// TIA Portal project "Inyectora_S7-1500" (V14)

(* hardware
DEVICE "S71500/ET200MP station_1"  S7-1500 station
   slot 0: "Perfil soporte_0"  Rack  6ES7 590-1***0-0AA0
   slot 1: "Inyectora"  CPU 1511-1 PN  6ES7 511-1AK01-0AB0  V2.1
      slot 3: "Display de la CPU_1"  6ES7591-1AA00-0AA0
   slot 2: "DI 16x24VDC BA_1"  DI 16x24VDC BA  6ES7 521-1BH10-0AA0  V1.0
   slot 3: "DQ 8x24VDC/2A HF_1"  DQ 8x24VDC/2A HF  6ES7 522-1BF00-0AB0  V2.1
   slot 4: "AI 8xU/I/RTD/TC ST_1"  AI 8xU/I/RTD/TC ST  6ES7 531-7KF00-0AB0  V2.1
   slot 5: "AI 8xU/I/RTD/TC ST_2"  AI 8xU/I/RTD/TC ST  6ES7 531-7KF00-0AB0  V2.1
   slot 6: "AI 8xU/I/RTD/TC ST_4"  AI 8xU/I/RTD/TC ST  6ES7 531-7KF00-0AB0  V2.1
   slot 7: "AI 8xU/I/RTD/TC ST_5"  AI 8xU/I/RTD/TC ST  6ES7 531-7KF00-0AB0  V2.1
   slot 8: "AQ 8xU/I HS_1"  AQ 8xU/I HS  6ES7 532-5HF00-0AB0  V2.1
   slot 9: "AQ 8xU/I HS_2"  AQ 8xU/I HS  6ES7 532-5HF00-0AB0  V2.1
*)

// ===== PLC "Inyectora"  CPU 1511-1 PN =====

VAR_GLOBAL   // PLC tag table "Tabla de variables estándar"
   "System_Byte" AT %MB1 : Byte;
   "FirstScan" AT %M1.0 : Bool;
   "DiagStatusUpdate" AT %M1.1 : Bool;
   "AlwaysTRUE" AT %M1.2 : Bool;
   "AlwaysFALSE" AT %M1.3 : Bool;
   "System_Byte(1)" AT %MB1 : Byte;
   "Clock_Byte" AT %MB0 : Byte;
   "Clock_10Hz" AT %M0.0 : Bool;
   "Clock_5Hz" AT %M0.1 : Bool;
   "Clock_2.5Hz" AT %M0.2 : Bool;
   "Clock_2Hz" AT %M0.3 : Bool;
   "Clock_1.25Hz" AT %M0.4 : Bool;
   "Clock_1Hz" AT %M0.5 : Bool;
   "Clock_0.625Hz" AT %M0.6 : Bool;
   "Clock_0.5Hz" AT %M0.7 : Bool;
   "DI_Selectora_Calentar" AT %I1.3 : Bool;   // Selectora 0=OFF; 1=ON
   "AQ_S_RETROCESO_CARRO" AT %QW104 : Int;
END_VAR

VAR_GLOBAL   // PLC tag table "DI"
   "DI_R_CARGA" AT %I0.2 : Bool;   // Recorridos de carga
   "DI_R_SUCCION" AT %I0.1 : Bool;   // Recorrido de succión
   "DI_S_PUERTA" AT %I0.0 : Bool;   // Seguridad de las puertas
   "DI_E_Local" AT %I0.3 : Bool;   // Parada de Emergencia desde el Tablero LOCAL
   "DI_E_Remoto" AT %I0.4 : Bool;   // Parada de Emergencia desde el Tablero Remoto
   "DI_Selectora_M" AT %I0.5 : Bool;   // Selectora MANUAL 0=OFF; 1=ON
   "DI_Selectora_S" AT %I0.6 : Bool;   // Selectora SEMIAUTOMATICO 0=OFF; 1=ON
   "DI_Selectora_A" AT %I0.7 : Bool;   // Selectora AUTOMATICO 0=OFF; 1=ON
   "DI_Arranque_L" AT %I1.0 : Bool;   // Boton de arranque del tablero LOCAL
   "DI_Parada_L" AT %I1.1 : Bool;   // Boton de parada del tablero LOCAL
   "DI_Selectora_LR" AT %I1.2 : Bool;   // Selectora 0=LOCAL; 1=REMOTO
END_VAR

VAR_GLOBAL   // PLC tag table "AI"
   "AI_P_HYD_INYECCION" AT %IW10 : Int;   // Presión Hidráulica de inyecc
   "AI_P_CE_MOLDE" AT %IW12 : Int;   // Presión de cierre de molde
   "AI_P_AP_MOLDE" AT %IW14 : Int;   // Presión de apertura de molde
   "AI_P_EXP_PIEZA" AT %IW16 : Int;   // Presión de expulsión de las piezas
   "AI_P_SUCCION" AT %IW18 : Int;   // Presión de succión
   "AI_P_MOV_CARRO" AT %IW20 : Int;   // Presión de movimiento carro
   "AI_P_GENERAL" AT %IW22 : Int;   // Presión general
   "AI_V_CARGA" AT %IW24 : Int;   // Velocidad de carga 0..100
   "AI_V_INYECCION" AT %IW30 : Int;   // Velocidad de inyección
   "AI_V_AP_MOLDE" AT %IW32 : Int;   // Velocidad de apertura de molde
   "AI_V_CE_MOLDE" AT %IW34 : Int;   // Velocidad de cierre de molde
   "AI_V_EXP_AVANCE" AT %IW36 : Int;   // Velocidad de expulsión avance
   "AI_V_EXP_RETROCESO" AT %IW38 : Int;   // Velocidad de expulsión retroceso
   "AI_V_CARRO" AT %IW40 : Int;   // Velocidad del carro
   "AI_V_SUCCION" AT %IW42 : Int;   // Velocidad de succión
   "AI_T_Z_ALIMENTACION" AT %IW44 : Int;   // Zona de Alimentación-real
   "T_Z_PLASTIFICACION" AT %IW90 : Int;   // Zona de Plastificación
   "T_Z_DOSIFICACION" AT %IW92 : Int;   // Zona de Dosifacion
   "T_Z_BOQUILLA" AT %IW94 : Int;   // Zona de Boquilla
   "T_MOLDE" AT %IW96 : Int;   // Temperatura del Molde
   "T_ACEITE_HYD" AT %IW98 : Int;   // Temperatura del Aceite Hidráulico
   "T_GABINETE" AT %IW100 : Int;   // Temperatura del Gabinete eléctrico
   "R_AV_INYECTOR" AT %IW102 : Int;   // Recorridos de avance inyector
   "R_AP_MOLDE" AT %IW104 : Int;   // Recorrido apertura del molde
   "AI_R_CE_MOLDE" AT %IW70 : Int;   // Recorrido cierre del molde
   "AI_R_CARRO" AT %IW72 : Int;   // Recorrido del carro
   "AI_R_EXPULSION" AT %IW74 : Int;   // Recorrido de la expulsión
END_VAR

VAR_GLOBAL   // PLC tag table "DQ"
   "DQ_VENTILADOR_GABINETE" AT %Q0.0 : Bool;
   "DQ_Z_ALIMENTACION" AT %Q0.1 : Bool;
   "DQ_Z_PLASTIFICACION" AT %Q0.2 : Bool;
   "DQ_Z_DOSIFICACION" AT %Q0.3 : Bool;
   "DQ_Z_BOQUILLA" AT %Q0.4 : Bool;
   "DQ_VENTILADOR" AT %Q0.5 : Bool;
END_VAR

VAR_GLOBAL   // PLC tag table "AQ"
   "AQ_S_INYECCION" AT %QW90 : Int;   // Solenoide de inyección
   "AQ_S_SUCCION" AT %QW92 : Int;   // Solenoide de succión
   "AQ_S_CARGA" AT %QW94 : Int;   // Solenoide de carga
   "AQ_S_EXPULSION" AT %QW96 : Int;   // Solenoide de Expulsión
   "AQ_S_AVANCE_CARRO" AT %QW98 : Int;   // Solenoide de movimiento de Carro
   "AQ_S_P_GENERAL" AT %QW100 : Int;   // Solenoide de presión General
   "AQ_S_R_CAUDAL" AT %QW102 : Int;   // Selenoide regulador de caudal
   "AQ_S_NOYO2" AT %QW110 : Int;   // Solenoide Noyo
   "AQ_S_NOYO3" AT %QW112 : Int;   // Solenoide Noyo
END_VAR

TYPE "Mediciones"
   STRUCT
      Medicion : Array[1..10] of Real;
   END_STRUCT;
END_TYPE

DATA_BLOCK "DB_Sistema"   // DB1
{ S7_Optimized_Access := 'TRUE' }
VERSION : 0.1
   VAR
      Lecturas : Struct   // Lecturas Procesadas
         Temperatura : Struct   // Lecturas de Temperatura, escaladas y normalizadas.
            Alimentacion : Real;   // Valor de Temperatura en la Zona de Alimentacion, ya normalizada y escalada.
            Plastificacion : Real;   // Valor de Temperatura en la Zona de Plastificacion, ya normalizada y escalada.
            Dosificacion : Real;   // Valor de Temperatura en la Zona de Dosificacion, ya normalizada y escalada.
            Boquilla : Real;   // Valor de Temperatura en la Zona de Boquilla, ya normalizada y escalada.
            Molde : Real;   // Valor de Temperatura del Molde, ya normalizada y escalada.
            Aceite : Real;   // Valor de Temperatura en el Aceite, ya normalizada y escalada.
            Gabinete : Real;   // Valor de Temperatura en el Gabinete, ya normalizada y escalada.
         END_STRUCT;
         Velocidad : Struct   // Lecturas de Velocidad, escalados y normalizados.
            Carga : Real;
            Inyeccion : Real;
            Apertura_Molde : Real;
            Cierre_Molde : Real;
            Expulsion_Avance : Real;
            Expulsion_Retroceso : Real;
            Carro : Real;
            Succion : Real;
         END_STRUCT;
         Recorrido : Struct   // Lecturas de Recorrido, escalados y normalizados.
            Avance_Inyector : Real;
            Apertura_Molde : Real;
            Cierre_Molde : Real;
            Carro : Real;
            Expulsion : Real;
         END_STRUCT;
         Presion : Struct   // Lecturas de Presiones, escaladas y normalizadas.
            Hidraulica_inyeccion : Real;
            Cierre_Molde : Real;
            Apertura_Molde : Real;
            Expulsion_Pieza : Real;
            Succion : Real;
            Movimiento_Carro : Real;
            General : Real;
            Seguridad_Molde : Real;
         END_STRUCT;
         Nivel_Tolva : Real;   // Lectura de Nivel, escalada y normalizada.
      END_STRUCT;
      Consigna : Struct   // Establecimiento de los Set Points
         Temperatura : Struct
            Alimentacion : Real;
            Plastificacion : Real;
            Dosificacion : Real;
            Boquilla : Real;
            Molde : Real;
            Aceite : Real;
            Gabinete : Real;
         END_STRUCT;
         Velocidad : Struct
            Carga : Real;
            Inyeccion : Real;
            Apertura_Molde : Real;
            Cierre_Molde : Real;
            Expulsion_Avance : Real;
            Expulsion_Retroceso : Real;
            Carro : Real;
            Succion : Real;
         END_STRUCT;
         Recorrido : Struct
            Avance_Inyector : Bool;
            Apertura_Molde : Bool;
            Cierre_Molde : Bool;
            Carro : Bool;
            Expulsion : Bool;
         END_STRUCT;
         Presion : Struct
            Hidraulica_inyeccion : Bool;
            Cierre_Molde : Bool;
            Apertura_Molde : Bool;
            Expulsion_Pieza : Bool;
            Succion : Bool;
            Movimiento_Carro : Bool;
            General : Bool;
            Seguridad_Molde : Bool;
         END_STRUCT;
         Tiempo : Struct
            Inyeccion : Real;
            Carga : Real;
            Curado : Real;
            Apertura_Molde : Real;
            Cierre_Molde : Real;
            Expulsion : Real;
            Retencion_Expulsion : Real;
            Reciclo : Real;
            Succion : Real;
            Carro : Real;
            Ciclo_Completo : Real;
         END_STRUCT;
      END_STRUCT;
      HMI : Struct   // Comandos del HMI
         CMD_Parada : Bool;   // Boton Parada HMI
         CMD_Arranque : Bool;   // Boton Arranque HMI
      END_STRUCT;
      Marcas : Struct   // Marcas para valores intermedios
         Selenoides : Struct
            Inyeccion : Bool;
            Succion : Bool;
            Carga : Bool;
            Expulsion : Bool;
            Avance_Carro : Bool;
            Retroceso_Carro : Bool;
            Presion_General : Bool;
            Regulador_Caudal : Bool;
            Noyo : Array[1..3] of Bool;
         END_STRUCT;
      END_STRUCT;
      Seguridad : Struct   // Marcas para control de seguridad
         Parada_Controlada : Bool;
         Parada_Emergencia : Bool;
      END_STRUCT;
      Paso : Array[1..10] of Bool;   // Marcas de pasos a seguir en la secuencia
   END_VAR
BEGIN
END_DATA_BLOCK

DATA_BLOCK "Valvula_Proporcional_1"   // DB5
{ S7_Optimized_Access := 'TRUE' }
VERSION : 0.1
// stored: InstanceOfName Valvula_Proporcional
"Valvula_Proporcional"
BEGIN
END_DATA_BLOCK

FUNCTION_BLOCK "Filtro"   // FB1, LAD
{ S7_Optimized_Access := 'TRUE' }
VERSION : 0.1
   VAR_INPUT
      Medicion : Real;
   END_VAR
   VAR_OUTPUT
      Valor_filtrado : Real;
   END_VAR
   VAR
      Mediciones : "Mediciones";
   END_VAR
   VAR_TEMP
      Sumatoria : Real;
   END_VAR
   VAR CONSTANT
      Divisior : Real := 10.0;
   END_VAR
BEGIN

REGION Network 1
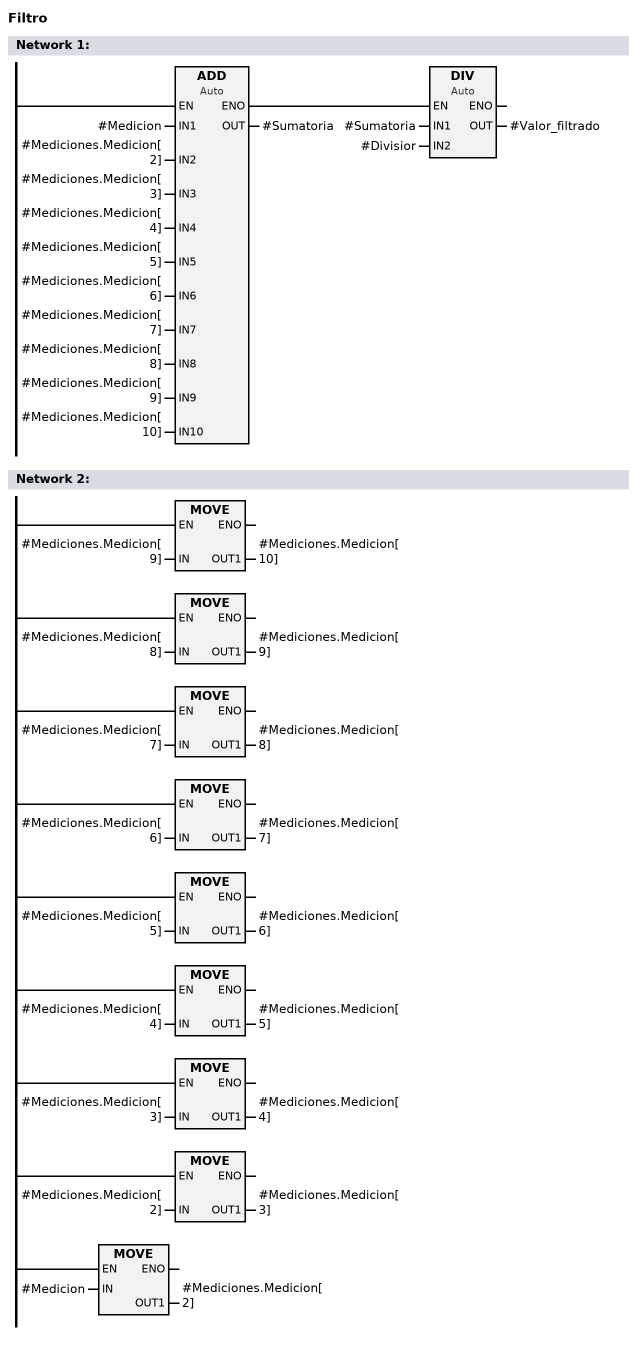
   RUNG wire#powerrail
      Add(in1 := #Medicion, in2 := #Mediciones.Medicion[2], in3 := #Mediciones.Medicion[3], in4 := #Mediciones.Medicion[4], in5 := #Mediciones.Medicion[5], in6 := #Mediciones.Medicion[6], in7 := #Mediciones.Medicion[7], in8 := #Mediciones.Medicion[8], in9 := #Mediciones.Medicion[9], in10 := #Mediciones.Medicion[10], out => #Sumatoria)
      Div(in1 := #Sumatoria, in2 := #Divisior, out => #Valor_filtrado)
   END_RUNG
   // the same network as SCL:
   #Sumatoria := #Medicion + #Mediciones.Medicion[2] + #Mediciones.Medicion[3] + #Mediciones.Medicion[4] + #Mediciones.Medicion[5] + #Mediciones.Medicion[6] + #Mediciones.Medicion[7] + #Mediciones.Medicion[8] + #Mediciones.Medicion[9] + #Mediciones.Medicion[10];
   #Valor_filtrado := #Sumatoria / #Divisior;
END_REGION

REGION Network 2
   RUNG wire#powerrail
      Move(in := #Mediciones.Medicion[9], out1 => #Mediciones.Medicion[10])
   END_RUNG
   RUNG wire#powerrail
      Move(in := #Mediciones.Medicion[8], out1 => #Mediciones.Medicion[9])
   END_RUNG
   RUNG wire#powerrail
      Move(in := #Mediciones.Medicion[7], out1 => #Mediciones.Medicion[8])
   END_RUNG
   RUNG wire#powerrail
      Move(in := #Mediciones.Medicion[6], out1 => #Mediciones.Medicion[7])
   END_RUNG
   RUNG wire#powerrail
      Move(in := #Mediciones.Medicion[5], out1 => #Mediciones.Medicion[6])
   END_RUNG
   RUNG wire#powerrail
      Move(in := #Mediciones.Medicion[4], out1 => #Mediciones.Medicion[5])
   END_RUNG
   RUNG wire#powerrail
      Move(in := #Mediciones.Medicion[3], out1 => #Mediciones.Medicion[4])
   END_RUNG
   RUNG wire#powerrail
      Move(in := #Mediciones.Medicion[2], out1 => #Mediciones.Medicion[3])
   END_RUNG
   RUNG wire#powerrail
      Move(in := #Medicion, out1 => #Mediciones.Medicion[2])
   END_RUNG
   // the same network as SCL:
   #Mediciones.Medicion[10] := #Mediciones.Medicion[9];
   #Mediciones.Medicion[9] := #Mediciones.Medicion[8];
   #Mediciones.Medicion[8] := #Mediciones.Medicion[7];
   #Mediciones.Medicion[7] := #Mediciones.Medicion[6];
   #Mediciones.Medicion[6] := #Mediciones.Medicion[5];
   #Mediciones.Medicion[5] := #Mediciones.Medicion[4];
   #Mediciones.Medicion[4] := #Mediciones.Medicion[3];
   #Mediciones.Medicion[3] := #Mediciones.Medicion[2];
   #Mediciones.Medicion[2] := #Medicion;
END_REGION
END_FUNCTION_BLOCK

FUNCTION_BLOCK "Valvula_Proporcional"   // FB2, LAD
{ S7_Optimized_Access := 'TRUE' }
VERSION : 0.1
   VAR_INPUT
      Consigna_Velocidad : Real;
      Posicion : Real;
   END_VAR
   VAR_OUTPUT
      Salida : Real;
   END_VAR
   VAR
      Captura_Posicion : Real;
   END_VAR
   VAR_TEMP
      PID_Salida : Real;
      Velocidad : Real;
      Porciento : Real;
   END_VAR
   VAR CONSTANT
      Divisor : Real := 0.01;   // La diferencia de tiempo es constante, se activa por una interrupcion ciclica
   END_VAR
BEGIN

REGION Network 1
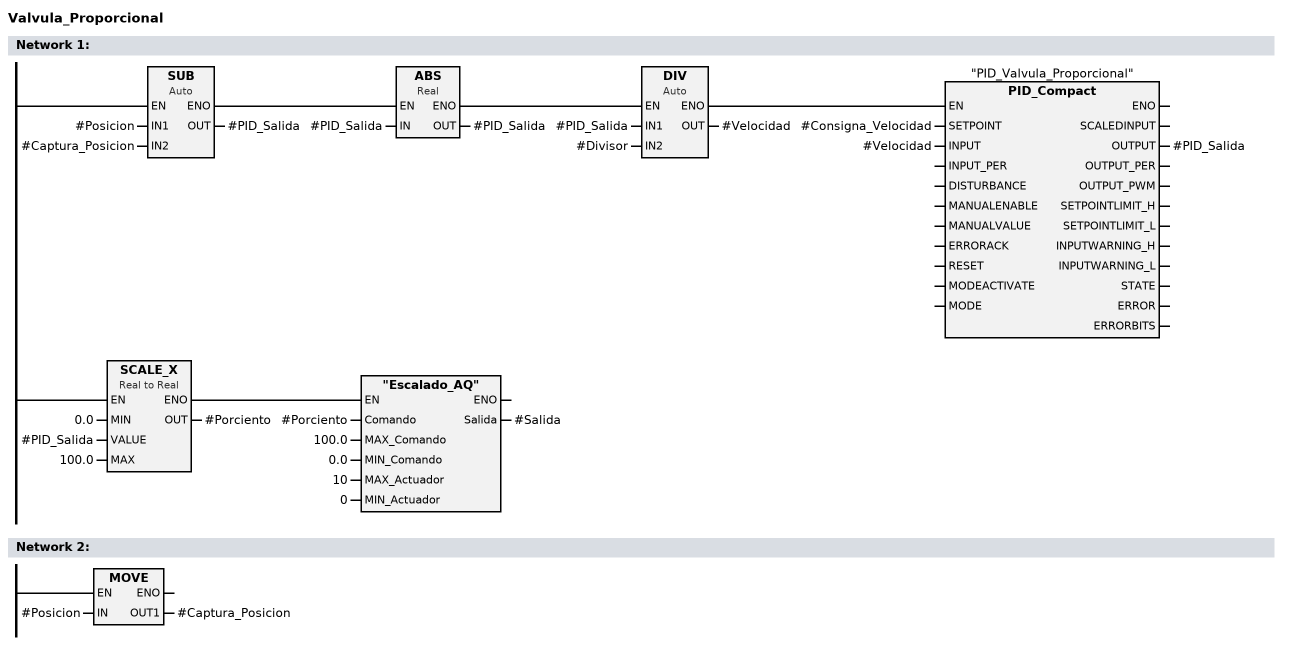
   #PID_Salida := #Posicion - #Captura_Posicion;
   #PID_Salida := ABS(#PID_Salida);
   #Velocidad := #PID_Salida / #Divisor;
   "PID_Valvula_Proporcional"(Setpoint := #Consigna_Velocidad, Input := #Velocidad, Output => #PID_Salida);   // PID_Compact
   #Porciento := SCALE_X(MIN := 0.0, VALUE := #PID_Salida, MAX := 100.0);
   "Escalado_AQ"(Comando := #Porciento,
                 MAX_Comando := 100.0,
                 MIN_Comando := 0.0,
                 MAX_Actuador := 10,
                 MIN_Actuador := 0,
                 Salida => #Salida);
END_REGION

REGION Network 2
   RUNG wire#powerrail
      Move(in := #Posicion, out1 => #Captura_Posicion)
   END_RUNG
   // the same network as SCL:
   #Captura_Posicion := #Posicion;
END_REGION
END_FUNCTION_BLOCK

FUNCTION "Seguridad" : Void   // FC1, LAD
{ S7_Optimized_Access := 'TRUE' }
VERSION : 0.1
BEGIN
END_FUNCTION

FUNCTION "Secuencia_Manual" : Void   // FC2, LAD
{ S7_Optimized_Access := 'TRUE' }
VERSION : 0.1
BEGIN
END_FUNCTION

FUNCTION "Escalado_AI" : Void   // FC3, LAD
TITLE = Escalado de las entradas Analogica
{ S7_Optimized_Access := 'TRUE' }
VERSION : 0.1
// 1. Normalizacion del valor obtenido por el sensor
//      a. El valor minimo del canal sera siempre 0. 
//      b. El valor maximo del canal lo obtendremos del datasheet del PLC.
//          Consultar Rangos de entrada analogica de tension/corriente
//          0..20mA / 4..20mA  --> 0..27648
//          0..10V  --> 0..27648
// 2. Escalado del valor normalizado
//       a. Minimo valor de lectura del sensor, nos lo da el fabricante.
//       b. Maximo valor de lectura del sensor.
   VAR_INPUT
      Sensor : Int;
      MAX_Sensor : Real;
      MIN_Sensor : Real;
      MAX_Canal : Int;
      MIN_Canal : Int;
   END_VAR
   VAR_OUTPUT
      Salida : Real;
   END_VAR
   VAR_TEMP
      Normalizado : Real;
   END_VAR
BEGIN

REGION Network 1
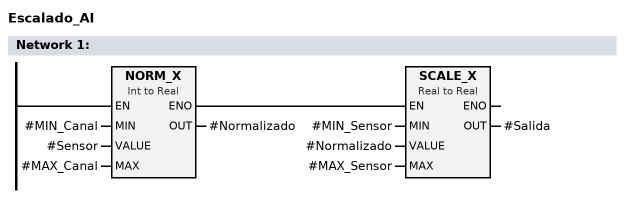
   RUNG wire#powerrail
      { S7_Templates := "[SrcType := Int, DestType := Real]" } Normalize(min := #MIN_Canal, value := #Sensor, max := #MAX_Canal, out => #Normalizado)
      { S7_Templates := "[SrcType := Real, DestType := Real]" } Scale(min := #MIN_Sensor, value := #Normalizado, max := #MAX_Sensor, out => #Salida)
   END_RUNG
   // the same network as SCL:
   #Normalizado := NORM_X(MIN := #MIN_Canal, VALUE := #Sensor, MAX := #MAX_Canal);
   #Salida := SCALE_X(MIN := #MIN_Sensor, VALUE := #Normalizado, MAX := #MAX_Sensor);
END_REGION
END_FUNCTION

FUNCTION "Escalado_AQ" : Void   // FC4, LAD
TITLE = Escalado de las salidas Analogicas
{ S7_Optimized_Access := 'TRUE' }
VERSION : 0.1
// 1. Normalizacion del valor seteado (comando)
//      a. El valor minimo del comando posible por el sistema a controlar. 
//      b. El valor maximo del comando es el posible por el sistema a controlar.
// Ejemplo: Motor de 0 a 600 RPM
// 2. Escalado del valor normalizado
//       a. Minimo valor del actuador producido por el Canal.
//       b. Maximo valor del actuador producido por el Canal
// .         Consultar Rangos de salida analogica de tension/corriente
//           0..20mA / 4..20mA  --> 0..27648
//           0..10V  --> 0..27648
   VAR_INPUT
      Comando : Real;
      MAX_Comando : Real;
      MIN_Comando : Real;
      MAX_Actuador : Int;
      MIN_Actuador : Int;
   END_VAR
   VAR_OUTPUT
      Salida : Int;
   END_VAR
   VAR_TEMP
      Nomalizado : Real;
   END_VAR
BEGIN

REGION Network 1
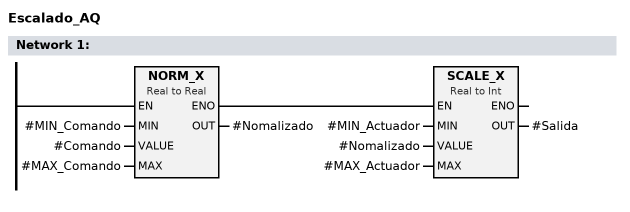
   RUNG wire#powerrail
      { S7_Templates := "[SrcType := Real, DestType := Real]" } Normalize(min := #MIN_Comando, value := #Comando, max := #MAX_Comando, out => #Nomalizado)
      { S7_Templates := "[SrcType := Real, DestType := Int]" } Scale(min := #MIN_Actuador, value := #Nomalizado, max := #MAX_Actuador, out => #Salida)
   END_RUNG
   // the same network as SCL:
   #Nomalizado := NORM_X(MIN := #MIN_Comando, VALUE := #Comando, MAX := #MAX_Comando);
   #Salida := SCALE_X(MIN := #MIN_Actuador, VALUE := #Nomalizado, MAX := #MAX_Actuador);
END_REGION
END_FUNCTION

FUNCTION "Secuencia_SemiAutomatica" : Void   // FC5, LAD
{ S7_Optimized_Access := 'TRUE' }
VERSION : 0.1
BEGIN
END_FUNCTION

FUNCTION "Secuencia_Automatica" : Void   // FC6, LAD
{ S7_Optimized_Access := 'TRUE' }
VERSION : 0.1
BEGIN
END_FUNCTION

FUNCTION "Lectura_Temperatura" : Void   // FC7, LAD
{ S7_Optimized_Access := 'TRUE' }
VERSION : 0.1
BEGIN
END_FUNCTION

FUNCTION "Lectura_Velocidad" : Void   // FC8, LAD
{ S7_Optimized_Access := 'TRUE' }
VERSION : 0.1
BEGIN
END_FUNCTION

FUNCTION "Lectura_Recorrido" : Void   // FC9, LAD
{ S7_Optimized_Access := 'TRUE' }
VERSION : 0.1
BEGIN
END_FUNCTION

FUNCTION "Lectura_Nivel" : Void   // FC10, LAD
{ S7_Optimized_Access := 'TRUE' }
VERSION : 0.1
BEGIN
END_FUNCTION

FUNCTION "Lectura_Presion" : Void   // FC11, LAD
{ S7_Optimized_Access := 'TRUE' }
VERSION : 0.1
BEGIN
END_FUNCTION

FUNCTION "Seleccion" : Void   // FC12, LAD
TITLE = Seleccion del Modo de Arranque y Secuencia (Por ahora solo en tablero)
{ S7_Optimized_Access := 'TRUE' }
VERSION : 0.1
// 1. Si se esta ejecutando una secuencia, la bobina NC de Paso[1] se abre e impide un cambio de secuencia en mitad del proceso.
// 2. Si se precionan los botones de Parada local o Remota, la bobina NC Parada_Controlada.
// 3. Si ocurrio un error en la secuencia, se activa la parada de emergencia.
// 4. Calentamos la maquina si la Selectora_Calentar esta en 1.
// 5. Si la selectora esta en Local no podremos arrancarla desde el HMI, solo se podra desde el boton en el tablero Local y viceversa  
// 6. Preguntamos si la temperatura de alimentacion es mayor a 200.0, si no es asi no podra arrancar la secuencia.
// 7. Para proteccion, si las salidas de la selectora estan haciendo contacto entre ellas no arrancara la secuencia.
   VAR_TEMP   // added for the SCL form of the ladder/FBD networks
      _w1 : Bool;
      _w2 : Bool;
   END_VAR
BEGIN

REGION Network 1
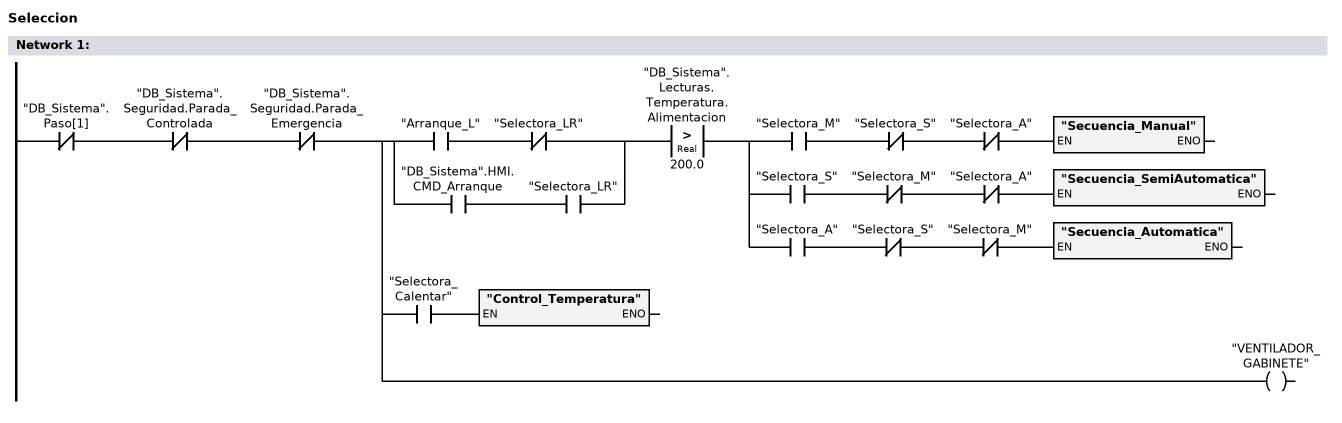
   RUNG wire#powerrail
      I_Contact( "DB_Sistema".Paso[1] )
      I_Contact( "DB_Sistema".Seguridad.Parada_Controlada )
      I_Contact( "DB_Sistema".Seguridad.Parada_Emergencia )
      wire#w1
      Contact( "Arranque_L" )
      I_Contact( "Selectora_LR" )
      wire#w2
      { S7_Templates := "SrcType := Real" } GT_Contact(in1 := "DB_Sistema".Lecturas.Temperatura.Alimentacion, in2 := 200.0)
      wire#w3
      Contact( "Selectora_M" )
      I_Contact( "Selectora_S" )
      I_Contact( "Selectora_A" )
      "Secuencia_Manual"()
   END_RUNG
   RUNG wire#w1
      Contact( "DB_Sistema".HMI.CMD_Arranque )
      Contact( "Selectora_LR" )
   END_RUNG wire#w2
   RUNG wire#w3
      Contact( "Selectora_S" )
      I_Contact( "Selectora_M" )
      I_Contact( "Selectora_A" )
      "Secuencia_SemiAutomatica"()
   END_RUNG
   RUNG wire#w3
      Contact( "Selectora_A" )
      I_Contact( "Selectora_S" )
      I_Contact( "Selectora_M" )
      "Secuencia_Automatica"()
   END_RUNG
   RUNG wire#w1
      Contact( "Selectora_Calentar" )
      "Control_Temperatura"()
   END_RUNG
   RUNG wire#w1
      Coil( "VENTILADOR_GABINETE" )
   END_RUNG
   // the same network as SCL:
   #_w1 := NOT "DB_Sistema".Paso[1] AND NOT "DB_Sistema".Seguridad.Parada_Controlada AND NOT "DB_Sistema".Seguridad.Parada_Emergencia;
   #_w2 := #_w1 AND (("Arranque_L" AND NOT "Selectora_LR") OR ("DB_Sistema".HMI.CMD_Arranque AND "Selectora_LR")) AND ("DB_Sistema".Lecturas.Temperatura.Alimentacion > 200.0);
   IF #_w2 AND "Selectora_M" AND NOT "Selectora_S" AND NOT "Selectora_A" THEN "Secuencia_Manual"(); END_IF;
   IF #_w2 AND "Selectora_S" AND NOT "Selectora_M" AND NOT "Selectora_A" THEN
       "Secuencia_SemiAutomatica"();
   END_IF;
   IF #_w2 AND "Selectora_A" AND NOT "Selectora_S" AND NOT "Selectora_M" THEN
       "Secuencia_Automatica"();
   END_IF;
   IF #_w1 AND "Selectora_Calentar" THEN "Control_Temperatura"(); END_IF;
   "VENTILADOR_GABINETE" := #_w1;
END_REGION
END_FUNCTION

FUNCTION "Control_Temperatura" : Void   // FC13, LAD
{ S7_Optimized_Access := 'TRUE' }
VERSION : 0.1
BEGIN

REGION Network 1
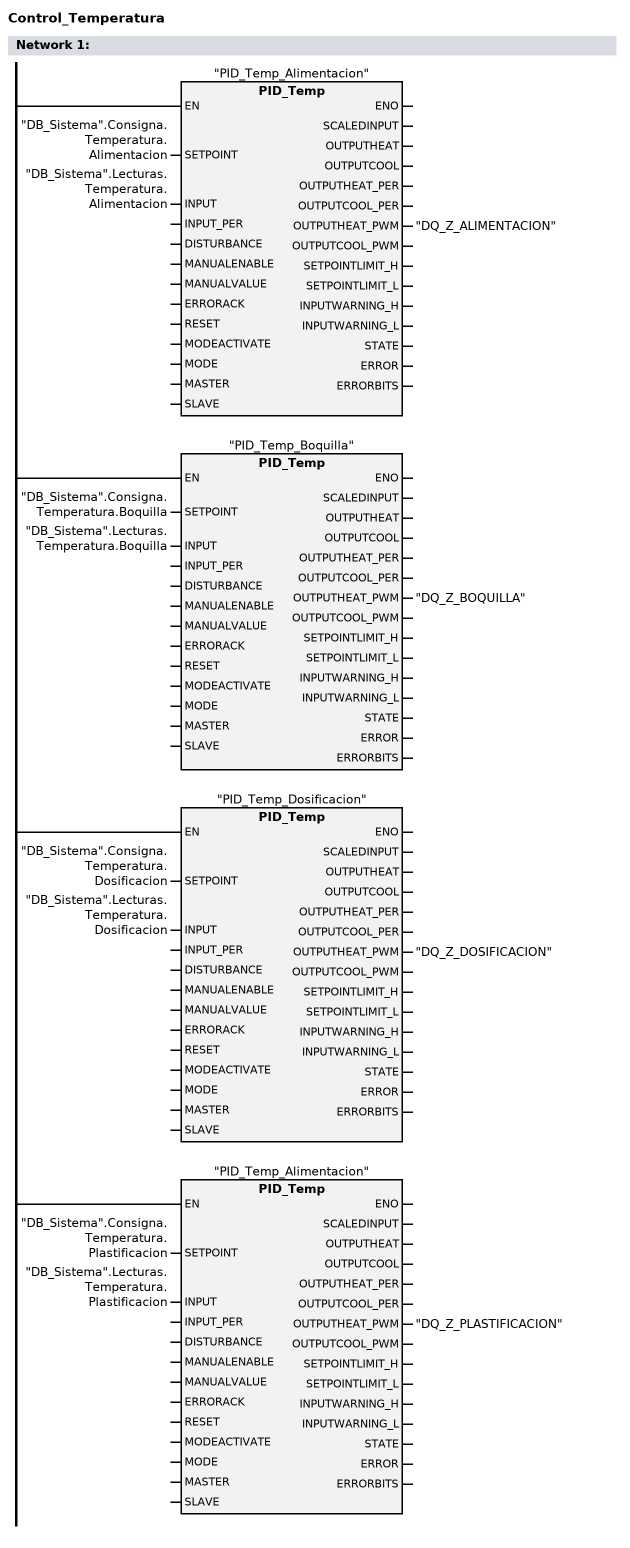
   "PID_Temp_Alimentacion"(Setpoint := "DB_Sistema".Consigna.Temperatura.Alimentacion,   // PID_Temp
                           Input := "DB_Sistema".Lecturas.Temperatura.Alimentacion,
                           OutputHeat_PWM => "DQ_Z_ALIMENTACION");
   "PID_Temp_Boquilla"(Setpoint := "DB_Sistema".Consigna.Temperatura.Boquilla,   // PID_Temp
                       Input := "DB_Sistema".Lecturas.Temperatura.Boquilla,
                       OutputHeat_PWM => "DQ_Z_BOQUILLA");
   "PID_Temp_Dosificacion"(Setpoint := "DB_Sistema".Consigna.Temperatura.Dosificacion,   // PID_Temp
                           Input := "DB_Sistema".Lecturas.Temperatura.Dosificacion,
                           OutputHeat_PWM => "DQ_Z_DOSIFICACION");
   "PID_Temp_Alimentacion"(Setpoint := "DB_Sistema".Consigna.Temperatura.Plastificacion,   // PID_Temp
                           Input := "DB_Sistema".Lecturas.Temperatura.Plastificacion,
                           OutputHeat_PWM => "DQ_Z_PLASTIFICACION");
END_REGION
END_FUNCTION

FUNCTION "Control_Selenoide" : Void   // FC14, LAD
{ S7_Optimized_Access := 'TRUE' }
VERSION : 0.1
BEGIN

REGION Network 1
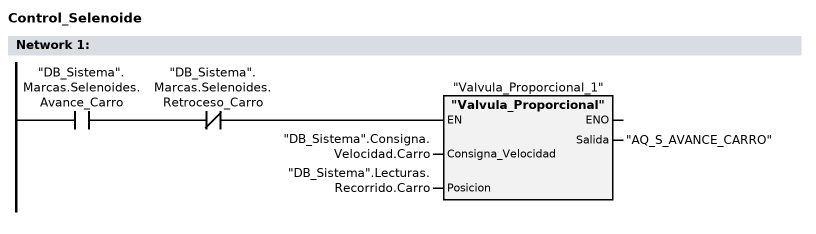
   RUNG wire#powerrail
      Contact( "DB_Sistema".Marcas.Selenoides.Avance_Carro )
      I_Contact( "DB_Sistema".Marcas.Selenoides.Retroceso_Carro )
      "Valvula_Proporcional_1"(Consigna_Velocidad := "DB_Sistema".Consigna.Velocidad.Carro, Posicion := "DB_Sistema".Lecturas.Recorrido.Carro, Salida => "AQ_S_AVANCE_CARRO")
   END_RUNG
   // the same network as SCL:
   IF "DB_Sistema".Marcas.Selenoides.Avance_Carro AND NOT "DB_Sistema".Marcas.Selenoides.Retroceso_Carro THEN
       "Valvula_Proporcional_1"(Consigna_Velocidad := "DB_Sistema".Consigna.Velocidad.Carro,   // "Valvula_Proporcional"
                               Posicion := "DB_Sistema".Lecturas.Recorrido.Carro,
                               Salida => "AQ_S_AVANCE_CARRO");
   END_IF;
END_REGION
END_FUNCTION

ORGANIZATION_BLOCK "Main"   // OB1, LAD, ProgramCycle
TITLE = "Main Program Sweep (Cycle)"
{ S7_Optimized_Access := 'TRUE' }
VERSION : 0.1
   VAR_INPUT
      Initial_Call : Bool;   // Initial call of this OB
      Remanence : Bool;   // =True, if remanent data are available
   END_VAR
BEGIN

REGION Network 1
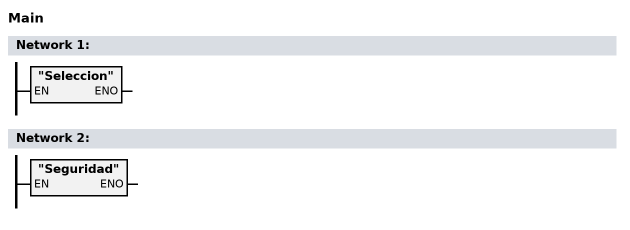
   RUNG wire#powerrail
      "Seleccion"()
   END_RUNG
   // the same network as SCL:
   "Seleccion"();
END_REGION

REGION Network 2
   RUNG wire#powerrail
      "Seguridad"()
   END_RUNG
   // the same network as SCL:
   "Seguridad"();
END_REGION
END_ORGANIZATION_BLOCK

ORGANIZATION_BLOCK "Interrupcion_Ciclica_Medicion"   // OB30, LAD, CyclicInterrupt
{ S7_Optimized_Access := 'TRUE' }
VERSION : 0.1
   VAR_INPUT
      Initial_Call : Bool;   // Initial call of this OB
      Event_Count : Int;   // Events discarded
   END_VAR
   VAR_TEMP   // added for the SCL form of the ladder/FBD networks
      _w1 : Bool;
   END_VAR
BEGIN

REGION Network 1
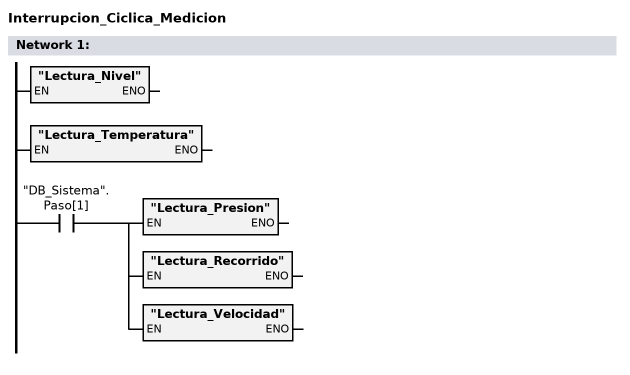
   RUNG wire#powerrail
      "Lectura_Nivel"()
   END_RUNG
   RUNG wire#powerrail
      "Lectura_Temperatura"()
   END_RUNG
   RUNG wire#powerrail
      Contact( "DB_Sistema".Paso[1] )
      wire#w1
      "Lectura_Presion"()
   END_RUNG
   RUNG wire#w1
      "Lectura_Recorrido"()
   END_RUNG
   RUNG wire#w1
      "Lectura_Velocidad"()
   END_RUNG
   // the same network as SCL:
   "Lectura_Nivel"();
   "Lectura_Temperatura"();
   #_w1 := "DB_Sistema".Paso[1];
   IF #_w1 THEN
       "Lectura_Presion"();
       "Lectura_Recorrido"();
       "Lectura_Velocidad"();
   END_IF;
END_REGION
END_ORGANIZATION_BLOCK

ORGANIZATION_BLOCK "Interrupcion_Ciclica_Control"   // OB31, LAD, CyclicInterrupt
{ S7_Optimized_Access := 'TRUE' }
VERSION : 0.1
   VAR_INPUT
      Initial_Call : Bool;   // Initial call of this OB
      Event_Count : Int;   // Events discarded
   END_VAR
BEGIN

REGION Network 1
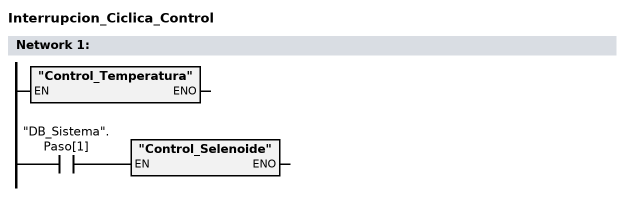
   RUNG wire#powerrail
      "Control_Temperatura"()
   END_RUNG
   RUNG wire#powerrail
      Contact( "DB_Sistema".Paso[1] )
      "Control_Selenoide"()
   END_RUNG
   // the same network as SCL:
   "Control_Temperatura"();
   IF "DB_Sistema".Paso[1] THEN "Control_Selenoide"(); END_IF;
END_REGION
END_ORGANIZATION_BLOCK